// TIA Portal V20 export
DATA_BLOCK "DB_ConveyorParameters"   // DB25
// stored: Access Published, MemoryReserve 100, Namespace PackedLine
   VAR
      Line : Struct
         PackedLine : Struct
            Conveyor : Array[_.minPackedLine.._.maxPackedLine] of "Global.ConveyorParameters";
         END_STRUCT;
      END_STRUCT;
   END_VAR
BEGIN
END_DATA_BLOCK
